INTERFACE IPmlStateMachine

METHOD getState : E_PMLState
VAR_INPUT
END_VAR
END_METHOD

METHOD PMLCommand : bool
VAR_INPUT
	Command : E_PMLCommand;
END_VAR
END_METHOD

METHOD StateComplete : BOOL
VAR_INPUT
END_VAR
END_METHOD

END_INTERFACE

(* stored: Version 1.1.0.1, ProductVersion 3.1.4024.9
   Itf IPmlStateMachine: Id {e9a51d04-2eb8-465c-a82b-7fd94f10d24e}
   Method getState: Id {c92b3ccb-9107-44d9-b563-97995e9d32ad}
   Method PMLCommand: Id {d2c71d0c-6799-4511-ad44-296dbc3c3f79}
   Method StateComplete: Id {d9c45e2d-bf3a-4f67-83c9-01bf887b92b0} *)
